// TIA Portal V18 export
// export: Created 2026-06-09T02:47:52.5257391Z, ExportSetting WithDefaults, DisplayName Totally Integrated Automation Portal, DisplayVersion V18, DisplayName TIA Portal Openness, DisplayVersion V18, DisplayName TIA Portal Version Control Interface, DisplayVersion V18, DisplayName STEP 7 Professional, DisplayVersion V18, DisplayName STEP 7 Safety, DisplayVersion V18, DisplayName WinCC Professional, DisplayVersion V18
VAR_GLOBAL   // PLC tag table "Nalewarka"
   start_nalewarka AT %M100.0 : Bool;
   stop_nalewarka AT %M100.1 : Bool;
   cz_pojemnosciowy AT %M200.0 : Bool;
   dozy AT %Q0.1 : Bool;
   tasma AT %Q0.0 : Bool;
   lampa AT %Q0.2 : Bool;
   wl_pomarancza AT %M212.0 : Bool;
   pomarancza AT %Q2.5 : Bool;
   wl_truskawka AT %M212.1 : Bool;
   truskawka AT %Q2.6 : Bool;
   cz_poz_napoju AT %M213.0 : Bool;
END_VAR
